VAR_GLOBAL
	// Boolean outputs
	bGreenLED AT %Q* : BOOL;
	bRedLED AT %Q* : BOOL;
	bEnableWinchValve AT %Q* : BOOL;
	bEnableCylValve AT %Q* : BOOL;
	
	// DINT outputs
	n_WinchValveOut AT %Q* : DINT;
	n_CylValveOut AT %Q* : DINT;
END_VAR

(* stored: Version 1.1.0.1, ProductVersion 3.1.4024.12
   GVL G_Output: Id {df32a59e-1940-47f1-8a1c-206918932020} *)
